{attribute addProperty BoxType "EL3208-0000-0017"}
{attribute addProperty Id "RTD_Inputs_ChannelAT %I*ARRAY[0..14] OF RTD_Inputs_Channel_17AE08DB256320WcStateAT %I*WcState_98A4DF7520.250InfoDataAT %I*InfoData_BC63D37F80100"}
{attribute addProperty CRC "3730341678"}
{attribute addProperty SizeInBites "338"}
{attribute addProperty SizeInBytes "42.25"}
TYPE EL3208_F6ED9915 :
STRUCT
	{attribute addProperty Name "RTD_Inputs_Channel"}
	RTD_Inputs_Channel : ARRAY[0..14] OF RTD_Inputs_Channel_17AE08DB;
	{attribute addProperty Name "WcState"}
	WcState : WcState_98A4DF75;
	{attribute addProperty Name "InfoData"}
	InfoData : InfoData_BC63D37F;
END_STRUCT
END_TYPE

(* stored: Version 1.2.0.0, ProductVersion 3.1.4024.9
   DUT EL3208_F6ED9915: Id {204e0a58-0e76-4751-8059-34df04fc2c8d} *)
